// TIA Portal V16 export
// export: Created 2021-09-08T12:46:09.4763272Z, ExportSetting WithDefaults, DisplayName Totally Integrated Automation Portal, DisplayVersion V16 Update 3, DisplayName TIA Portal Version Control Interface, DisplayVersion V16 Update 2, DisplayName TIA Portal Openness, DisplayVersion V16 Update 3, DisplayName TIA Portal Teamcenter Gateway, DisplayVersion V16, DisplayName STEP 7 Professional, DisplayVersion V16 Update 3, DisplayName STEP 7 Safety, DisplayVersion V16, DisplayName WinCC Advanced, DisplayVersion V16 Update 3
FUNCTION "setFlags" : Void   // FC2, FBD
{ S7_Optimized_Access := 'TRUE' }
VERSION : 0.1
// stored: AutoNumber true, IsIECCheckEnabled false, SetENOAutomatically false, UDAEnableTagReadback false
   VAR_INPUT
      enCondition : Bool;
      condition : Bool;
      setTimerVal : Real;
   END_VAR
   VAR_IN_OUT
      curFlag : Bool;
      mainFlag : Bool;
      timerVal : Real;
   END_VAR
BEGIN

REGION Network 1 (SCL)

   #curFlag := #enCondition AND #condition;

   IF NOT #curFlag THEN
       #timerVal := 0;
   END_IF;

   IF #curFlag AND #timerVal < #setTimerVal THEN
       #timerVal += 0.1;
   END_IF;

   IF #timerVal >= #setTimerVal THEN
       #mainFlag := TRUE;
   END_IF;
END_REGION
END_FUNCTION
